// Contains tests that verify the XmlControl function block methods
FUNCTION_BLOCK FB_TestXUnitPublisher EXTENDS TcUnit.FB_TestSuite

Test_EscapedFailedMessage();
Test_EscapedFunctionName();

METHOD PRIVATE Test_EscapedFailedMessage
TEST('Test_EscapedFailedMessage');

AssertTrue(FALSE, 'This "string" <should> be $'escaped$' & parsed properly');

TEST_FINISHED();
END_METHOD

METHOD PRIVATE Test_EscapedFunctionName
TEST('Test_EscapedFunctionName$'"<>&');

TEST_FINISHED();
END_METHOD

END_FUNCTION_BLOCK

(* stored: Version 1.1.0.1
   POU FB_TestXUnitPublisher: Id {c7819ac2-5de4-4840-89ae-815e54b5cb69}, SpecialFunc None
   Method Test_EscapedFailedMessage: Id {8aca4c27-6db1-484c-a76f-a529f691497e}
   Method Test_EscapedFunctionName: Id {da2058a6-4b6f-43f7-8364-e0cf3494d96b} *)
